FUNCTION Matrix_Scale : BOOL
VAR_IN_OUT
	M : Matrix;
END_VAR
VAR_INPUT
	Scalar : LREAL;
END_VAR

VAR
	I : UINT;
END_VAR

Matrix_Scale := TRUE;

IF M.IsEmpty THEN
	RETURN;
END_IF

FOR I := 0 TO M.Length-1 DO
	M.SetI(I,Scalar * M.GetI(I));
END_FOR

END_FUNCTION

(* stored: Version 1.1.0.1, ProductVersion 3.1.4024.9
   POU Matrix_Scale: Id {0a70bdcb-e9cf-0eec-2ebf-e6289b9019aa}, SpecialFunc None *)
